// TIA Portal V19 export
TYPE "LEXCHANGETRAY_typeConstraintWorkstationIoSignalContronNodeMonitoring"
// simulated: Bool
// hookClawCylinderWorkPositionDetection2: Bool
// slideCylinderMedianPositionDetection1: Bool
// slideCylinderWorkPositionDetection1: Bool
// motorConstraintPot2: Bool
// motorConstraintNot2: Bool
// motorConstraintPot1: Bool
// motorConstraintOrg2: Bool
// hookClawCylinderWorkPositionDetection1: Bool
// hookClawCylinderHomePositionDetection1: Bool
// pressureGaugeSetValueDetection2_2: Bool
// motorConstraintNot1: Bool
// slideCylinderHomePositionDetection1: Bool
// motorConstraintOrg1: Bool
// slideCylinderHomePositionDetection2: Bool
// pressureGaugeSetValueDetection1_2: Bool
// pressureGaugeSetValueDetection2_1: Bool
// slideCylinderWorkPositionDetection2: Bool
// hookClawCylinderHomePositionDetection2: Bool
// pressureGaugeSetValueDetection1_1: Bool
// slideCylinderMedianPositionDetection2: Bool
// stored: Access Published
   STRUCT
      simulated : Bool;
      hookClawCylinderWorkPositionDetection2 : Bool;
      slideCylinderMedianPositionDetection1 : Bool;
      slideCylinderWorkPositionDetection1 : Bool;
      motorConstraintPot2 : Bool;
      motorConstraintNot2 : Bool;
      motorConstraintPot1 : Bool;
      motorConstraintOrg2 : Bool;
      hookClawCylinderWorkPositionDetection1 : Bool;
      hookClawCylinderHomePositionDetection1 : Bool;
      pressureGaugeSetValueDetection2_2 : Bool;
      motorConstraintNot1 : Bool;
      slideCylinderHomePositionDetection1 : Bool;
      motorConstraintOrg1 : Bool;
      slideCylinderHomePositionDetection2 : Bool;
      pressureGaugeSetValueDetection1_2 : Bool;
      pressureGaugeSetValueDetection2_1 : Bool;
      slideCylinderWorkPositionDetection2 : Bool;
      hookClawCylinderHomePositionDetection2 : Bool;
      pressureGaugeSetValueDetection1_1 : Bool;
      slideCylinderMedianPositionDetection2 : Bool;
   END_STRUCT;
END_TYPE
